TYPE LEDControl :
STRUCT
	execute 	: BIT;
	send		: BIT;
	update		: BIT;
	command		: USINT;(*LEDCommands*)
	index 		: UINT;
	length		: UINT;
	parameter	: UINT;
	color 		: LEDColor;
END_STRUCT
END_TYPE

(* stored: Version 1.1.0.1, ProductVersion 3.1.4026.18
   DUT LEDControl: Id {bd6e9f6e-7679-4950-a9dd-4884ff50972a} *)
